// TwinCAT 3 PLC project Untitled1
// ProgramVersion: 3.1.4024.0
// libraries:
//   Tc2_ControllerToolbox, * (Beckhoff Automation GmbH)
//   Tc2_MC2, * (Beckhoff Automation GmbH)
//   Tc2_Standard, * (Beckhoff Automation GmbH)
//   Tc2_System, * (Beckhoff Automation GmbH)
//   Tc3_Module, * (Beckhoff Automation GmbH)
// project tree:
//   / PlcTask.TcTTO
//   POUs/ MAIN.TcPOU, PRG_Motion.TcPOU, PRG_TempControl.TcPOU
// real-time tasks:
//   TASK PlcTask: cycle T#10ms, priority 20, ADS port 350

CONFIGURATION Untitled1
    RESOURCE PLC ON TwinCAT3
        TASK PlcTask(INTERVAL := T#10ms, PRIORITY := 20);
        PROGRAM MAIN WITH PlcTask : MAIN;
    END_RESOURCE
END_CONFIGURATION

// ---- POUs/MAIN.TcPOU
PROGRAM MAIN
VAR
	Counter	:UDINT;
END_VAR

Counter:=Counter+1;
PRG_Motion();

PRG_TempControl();

END_PROGRAM

// ---- POUs/PRG_Motion.TcPOU
PROGRAM PRG_Motion
VAR
	Axis1		:AXIS_REF;
	Power		:MC_Power;
	MoveVelo	:MC_MoveVelocity;
	TriggerMove	:BOOL;
END_VAR

Power(
	Axis			:=Axis1 , 
	Enable			:=TRUE , 
	Enable_Positive	:=TRUE , 
	Enable_Negative	:=TRUE , 
	Override		:=100.0);
	
	
MoveVelo(
	Axis			:=Axis1 , 
	Execute			:=TriggerMove , 
	Velocity		:=1000.0 , 
	Acceleration	:=5000.0 , 
	Deceleration	:=5000.0 , 
	Jerk			:=10000.0 , 
	Direction		:=MC_Direction.MC_Positive_Direction);

END_PROGRAM

// ---- POUs/PRG_TempControl.TcPOU
PROGRAM PRG_TempControl
VAR
	SetPoint			: LREAL := 100;
	ActualTemp	AT %I*	: LREAL;
	Output		AT %Q*	: LREAL;
	fbPID				: FB_CTRL_PID;
	PID_Params			: ST_CTRL_PID_PARAMS := (tCtrlCycleTime	:= TIME#10ms,
												tTaskCycleTime	:= TIME#10ms,
												fKp				:= 10,
												tTn				:= TIME#100ms,
												tTv				:= TIME#45ms,
												tTd				:= TIME#1ms);
END_VAR

fbPID(fSetpointValue := SetPoint,
	fActualValue	:= ActualTemp,
	eMode			:= E_CTRL_MODE.eCTRL_MODE_ACTIVE,
	fOut			=> Output,
	stParams		:= PID_Params);

END_PROGRAM
